PROGRAM LightsON
VAR
END_VAR

IF GVL.AlarmON THEN
	GVL.LightsON := TRUE;
ELSE
	GVL.LightsON := FALSE;
END_IF

END_PROGRAM

(* stored: Version 1.1.0.1, ProductVersion 3.1.4024.12
   POU LightsON: Id {05eb1e63-91b5-433c-9b62-b9f70f8ec3be}, SpecialFunc None *)
